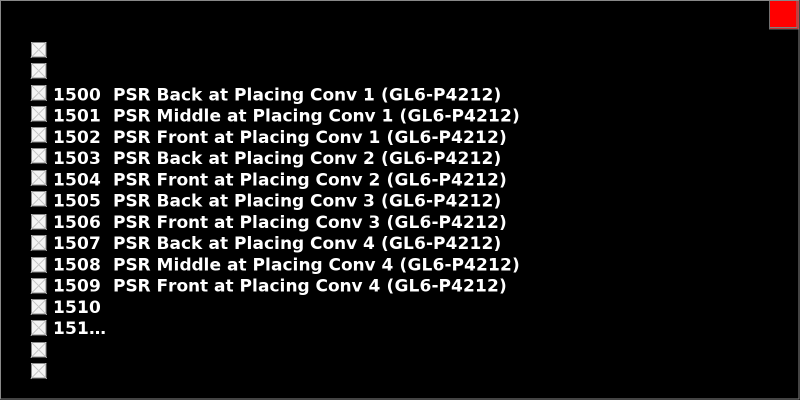
VISUALIZATION P1_DI4  // 800x400, background image 
    ImageSwitcher (31,42 15x15), variable: InputOutput_GVL.xIn1500, behaviour: TOGGLE
    Label (50,16 625x391), "1500 PSR Back at Placing Conv 1 (GL6-P4212) 1501 PSR Middle at Placing Conv 1 (GL6-P4212) 1502 PSR Front at Placing Conv 1 (GL6-P4212) 1503 PSR Back at Placing Conv 2 (GL6-P4212) 1504 PSR Front at Placing Conv 2 (GL6-P4212) 1505 PSR Back at Placing Conv 3 (GL6-P4212) 1506 PSR Front at Placing Conv 3 (GL6-P4212) 1507 PSR Back at Placing Conv 4 (GL6-P4212) 1508 PSR Middle at Placing Conv 4 (GL6-P4212) 1509 PSR Front at Placing Conv 4 (GL6-P4212) 1510 1511 1512 1513 1514 1515"
    ImageSwitcher (31,63 15x15), variable: InputOutput_GVL.xIn1501, behaviour: TOGGLE
    ImageSwitcher (31,85 15x15), variable: InputOutput_GVL.xIn1502, behaviour: TOGGLE
    ImageSwitcher (31,106 15x15), variable: InputOutput_GVL.xIn1503, behaviour: TOGGLE
    ImageSwitcher (31,127 15x15), variable: InputOutput_GVL.xIn1504, behaviour: TOGGLE
    ImageSwitcher (31,148 15x15), variable: InputOutput_GVL.xIn1505, behaviour: TOGGLE
    ImageSwitcher (31,170 15x15), variable: InputOutput_GVL.xIn1506, behaviour: TOGGLE
    ImageSwitcher (31,191 15x15), variable: InputOutput_GVL.xIn1507, behaviour: TOGGLE
    ImageSwitcher (31,214 15x15), variable: InputOutput_GVL.xIn1508, behaviour: TOGGLE
    ImageSwitcher (31,235 15x15), variable: InputOutput_GVL.xIn1509, behaviour: TOGGLE
    ImageSwitcher (31,257 15x15), variable: InputOutput_GVL.xIn1510, behaviour: TOGGLE
    ImageSwitcher (31,278 15x15), variable: InputOutput_GVL.xIn1511, behaviour: TOGGLE
    ImageSwitcher (31,299 15x15), variable: InputOutput_GVL.xIn1512, behaviour: TOGGLE
    ImageSwitcher (31,320 15x15), variable: InputOutput_GVL.xIn1513, behaviour: TOGGLE
    ImageSwitcher (31,342 15x15), variable: InputOutput_GVL.xIn1514, behaviour: TOGGLE
    ImageSwitcher (31,363 15x15), variable: InputOutput_GVL.xIn1515, behaviour: TOGGLE
    Button (769,-1 30x30), image: VisuSymbols.Symbols.Wrong
        OnMouseClick: CloseDialog Dialog=P1_DI4, Result=OK, NumpadKeypadSet=True
END_VISUALIZATION

(* stored: Version 1.1.0.1, ProductVersion 3.1.4024.12
   Visu P1_DI4: Id {dbce4a39-07f8-44aa-9070-c86025a19824} *)
